FUNCTION F_SetBeamParams : ST_BeamParams
VAR_INPUT
	fAtt	:	REAL := 100;
	fPP_mJ: REAL := 0;
	neVRange	:	WORD := 0;
	nRate	:	UDINT := 0;
END_VAR
VAR
	BeamParams	:	ST_BeamParams;
	
END_VAR

BeamParams.fAtt := LIMIT(0,fAtt,100);
BeamParams.fPP_mJ := LIMIT(0,fPP_mJ,20);
BeamParams.neVRange := neVRange;
BeamParams.nRate	:= MIN(nRate,1000000);

F_SetBeamParams	:= BeamParams;

END_FUNCTION

(* stored: Version 1.1.0.1, ProductVersion 3.1.4024.0
   POU F_SetBeamParams: Id {4c1793f1-8a27-0a2c-0990-5356f1b410e4}, SpecialFunc None *)
